Universal Robots PolyScope program: cobot_de_soudure_V2.2_GAPE.urp

Program cobot_de_soudure_V2.2_GAPE (installation=Cobot_de_soudure_V2.1_GAPE directory=/programs/Soudure 2023_03_27/V2.1 createdIn=5.9.4.1031232 lastSavedIn=5.11.9.1010452 robotSerialNumber=20225200921)
Calibrated DH parameters: a=[-0.00003, -0.368557, -0.560435, 0, -0.000026, 0]; d=[0.180818, -449.783649, 477.665205, -27.707784, 0.119652, 0.115612]; alpha=[1.571383, 0.001086, 0.003988, 1.568685, -1.571248, 0]; deltaTheta=[-0.000001, -0.924567, 7.403594, -0.195847, 0.000002, 0]
InitVariablesNode variables(variable(name=Test_Gaz, expression=False), variable(name=Test_Job, expression=False), variable(name=Test_Ordre_Mar, expression=False), variable(name=Valide_Gaz, expression=False), variable(name=fin_soud, expression=1), variable(name=secu_d, expression=0), variable(name=secu_g, expression=0), variable(name=timer_ret_gaz, expression=0))
BeforeStart
  Folder fonctions
    Folder Init [hidden by the author, left out]
    Folder Diverses
      Script file /programs/Soudure 2023_03_27/V2.1/scripts/Diverses/close_popup.script
        | #fermeture popup
        | 
        | def close_popup():
        | 	closepop = "close popup"
        |     	socket_send_string(closepop,"internal")
        |     	socket_send_byte(10,"internal")
        |     	socket_close()
        | 
        | 	closepop = "close popup"
        |     	socket_send_string(closepop,"internal")
        |     	socket_send_byte(10,"internal")
        |     	socket_close()
        | 	return(False)
        | end
      Script file /programs/Soudure 2023_03_27/V2.1/scripts/Diverses/debut_soud.script
        | def fun_debut_soudure():
        |     Valide_Gaz = False
        |     if  ((Test_Ordre_Mar == False) and (Test_Job == False)):
        |         Arc_On = True
        |         Test_Gaz = True
        |     end
        | end
      Script file /programs/Soudure 2023_03_27/V2.1/scripts/Diverses/fin_soudure.script
        | def fin_soudure():
        |         Arc_On = False
        |         Test_Gaz = False
        |         Test_Job = True
        |         Test_Ordre_Mar = True
        | end
      Script file /programs/Soudure 2023_03_27/V2.1/scripts/Diverses/fun_demande().script
        | #demande nombre soudures par type (compris entre 0 et 6)
        | 
        | def fun_demande(type):
        | 	if (1==type):
        | 		soudure = "point"					#si type = 1, la demande sera sur une soudure point
        | 	elif (2==type):
        | 		soudure = "lineaire"				#si type = 2, la demande sera sur une soudure linéaire
        | 	elif (3==type):
        | 		soudure = "arc de cercle"			#si type = 3, la demande sera sur une soudure arc de cercle
        | 	elif (4==type):
        | 		soudure = "cercle"					#si type = 4, la demande sera sur une soudure cercle
        | 	else :
        | 		return(False)
        | 	end
        | 
        | nb_soud = request_integer_from_primary_client("nombre de soudure(s) "+ soudure + " ?")			#la demande
        | 	if (nb_soud >6):																									#si la reponse est superieur a 6
        | 		popup1 = "popup le robot ne peut pas effectuer plus de 6 soudures "+ soudure + " sur la même pièce, réessayer."	#popup
        | 		socket_open("127.0.0.1",29999,"internal") # open internal socket
        | 
        | 		socket_send_line(popup1,"internal")         #Affichage Popup
        | 
        | 		socket_send_byte(10,"internal")
        | 		sleep(5.0)
        | 		closepop = "close popup"					#fermer popup
        | 		socket_send_string(closepop,"internal")
        | 		socket_send_byte(10,"internal")
        | 		socket_close()
        | 
        | 		while(nb_soud >6):
        | 			nb_soud = request_integer_from_primary_client("nombre de soudure(s) "+ soudure + " ? (compris entre 0 et 6 ;)")	#on redemande tant que le nombre est superieur a 6
        | 		end
        | end
        | return(nb_soud)        #on retourne le nombre de soudure à effectuer dans le type
        | end
      Script file /programs/Soudure 2023_03_27/V2.1/scripts/Diverses/fun_demande_job.script
        | #demande le job à utiliser (mode de soudure régler sur le poste à souder) (compris entre 0 et 3, pour 1 et 4 sur le poste a souder)
        | def fun_demande_job(type):
        | 	if (1==type):
        | 		soudure = "point"
        | 	elif (2==type):
        | 		soudure = "lineaire"
        | 	elif (3==type):
        | 		soudure = "arc de cercle"
        | 	elif (4==type):
        | 		soudure = "cercle"
        | 	else :
        | 		return(False)
        | 	end
        | 
        |   job = request_integer_from_primary_client("Mode du poste à souder pour soudure : "+ soudure + " ? [1-4]")
        |   job = job-1 #adapter la saisie aux besoins du code
        | 
        |   while ((job!=0) and (job!=1) and (job!=2) and (job!=3)): #reboucler si mauvaise saisie
        | 	  job = request_integer_from_primary_client("Mode du poste à souder pour soudure : "+ soudure + " ? [1-4]")
        |       job = job-1 #adapter la saisie aux besoins du code
        |   end
        | 
        | return(job)
        | end
      Script file /programs/Soudure 2023_03_27/V2.1/scripts/Diverses/fun_demande_type_soudure.script
        | #demande le type de soudure à enregistrer (entre 1 et 5)
        | def fun_demande_type_soudure():
        | 
        | 	reponse = request_integer_from_primary_client("1->POINT     2->LINEAIRE    3->ARC    4->CERCLE  5->FIN")
        | 
        |     if ((reponse == 0) or (reponse > 5)):
        |         reponse = 5
        |     end
        | 
        | return(reponse)
        | end
      Script file /programs/Soudure 2023_03_27/V2.1/scripts/Diverses/fun_demande_vit.script
        | #demande nombre soudures par type (compris entre 0 et 6)
        | def fun_demande_vit(type):
        | 	if (1==type):
        | 		soudure = "point"
        | 	elif (2==type):
        | 		soudure = "lineaire"
        | 	elif (3==type):
        | 		soudure = "arc de cercle"
        | 	elif (4==type):
        | 		soudure = "cercle"
        | 	else :
        | 		return(False)
        | 	end
        | 
        | vit_soud = request_float_from_primary_client("vitesse de la soudure "+ soudure + " ? (mm/s)")
        | 	#if (vit_soud >6):
        | 	#	popup1 = "popup le robot ne peut pas effectuer plus de 6 soudures "+ soudure + " sur la même pièce, réessayer."
        | 	#	socket_open("127.0.0.1",29999,"internal") # open internal socket
        | 
        | 	#	socket_send_line(popup1,"internal")         #Affichage Popup
        | 
        | 	#	socket_send_byte(10,"internal")
        | 	#	sleep(5.0)
        | 	#	closepop = "close popup"
        | 	#	socket_send_string(closepop,"internal")
        | 	#	socket_send_byte(10,"internal")
        | 	#	socket_close()
        | 
        | 	#	while(vit_soud >6):
        | 	#		vit_soud = request_integer_from_primary_client("nombre de soudure(s) "+ soudure + " ? (compris entre 0 et 6 ;)")
        | 	#	end
        | #end
        | return(vit_soud/1000)
        | end
      Script file /programs/Soudure 2023_03_27/V2.1/scripts/Diverses/fun_front_down.script
        | #attente front montant sur add_bp
        | 
        | def fun_front_do(add_bp):
        | bp = get_digital_in(add_bp)
        |     while not bp :
        |         bp = get_digital_in(add_bp)    #dans la boucle tant que l'entrée add_bp est a 1
        |         #attente relachement bouton
        |    end
        | 
        |     while bp :                              #dans la boucle tant que l'entrée add_bp est a 0
        |         bp = get_digital_in(add_bp)
        |         #attente
        |     end
        | 
        |     #while not bp :
        |            #bp = get_digital_in(add_bp)    #dans la boucle tant que l'entrée add_bp est a 1
        |      #end
        | 
        |     return(False)
        | end
      Script file /programs/Soudure 2023_03_27/V2.1/scripts/Diverses/fun_front_up.script
        | #attente front montant sur add_bp
        | 
        | def fun_front_up(add_bp):
        | bp = get_digital_in(add_bp)
        |     while bp :
        |         bp = get_digital_in(add_bp)    #dans la boucle tant que l'entrée add_bp est a 1
        |         #attente relachement bouton
        |     end
        | 
        |     while not bp :                              #dans la boucle tant que l'entrée add_bp est a 0
        |         bp = get_digital_in(add_bp)
        |         #attente
        |     end
        |     return(False)
        | end
      Script file /programs/Soudure 2023_03_27/V2.1/scripts/Diverses/fun_popup_soud().script
        | #ouvre un pop-up "configuration soudure (type_soud) n°(num_soud): placer le robot (etape_soud) et valider la position. (bp_cobot)". fermeture popup a l'aide de close_popup()
        | #pour la definition de la fonction :
        |     #etape :
        |     #   1 : approche
        |     #   2 : depart
        |     #   3 : premier quart
        |     #   4 : milieu
        |     #   5 : trois-quart
        |     #   6 : fin
        |     #   7 : retrait
        | 
        |     #type :
        |     #   1 : soudure point
        |     #   2 : soudure lineaire
        |     #   3 : soudure arc de cercle
        |     #   4 : soudure cercle
        |     #   5 : plus de soudure
        |     #num : i, j, k ou l correspondant au numero de la soudure ( i pour type = 1, j pour type = 2, k pour type = 3, l pour type = 4)
        | 
        | def fun_popup_soud(etape, type, num):
        | 
        |     switch_1 = etape
        |     switch_2 = type
        |         ##############################################################################
        | 
        |     ####################### POPUP-approche #######################################
        | 
        | ##############################################################################
        |     #switch etape
        |     if (1 == switch_1) : #point d'approche
        |         etape_soud = " en APPROCHE"
        |         #switch type
        |         if (1 == switch_2) : #soudure point
        |             type_soud = "point"
        | 
        |        elif (2 == switch_2) : #soudure lineaire
        |             type_soud = "lineaire"
        | 
        |         elif (3 == switch_2) : #soudure arc de cerlce
        |             type_soud = "arc de cercle"
        | 
        |         elif (4 == switch_2) : #soudure cercle
        |            type_soud = "cercle"
        | 
        |         else :
        |             return (False)
        |         end
        | 
        |         ##############################################################################
        | 
        |     ####################### POPUP-debut ##########################################
        | 
        | ##############################################################################
        | 
        |     elif (2 == switch_1): #point de soudure/debut
        |         #switch type
        |         if (1 == switch_2) : #soudure point
        |            etape_soud = "sur le POINT"
        |             type_soud = "point"
        | 
        |         elif (2 == switch_2): #soudure lineaire
        |             etape_soud = "sur le DEBUT"
        |             type_soud = "lineaire"
        | 
        |         elif (3 == switch_2) : #soudure arc de cerlce
        |             etape_soud = "sur le DEBUT"
        |             type_soud = "arc de cercle"
        | 
        |         elif (4 == switch_2) : #soudure cercle
        |             etape_soud = "sur le DEBUT"
        |            type_soud = "cercle"
        | 
        |         else :
        |             return (False)
        |         end
        | 
        |         ##############################################################################
        | 
        |     ####################### POPUP-quart ##########################################
        | 
        | ##############################################################################
        | 
        |     elif (3 == switch_1): #point de quart
        |         etape_soud = "sur 1er QUART"
        |         #switch type
        |         if (4 == switch_2) : #soudure cercle
        |             type_soud = "cercle"
        |         end
        | 
        |         ##############################################################################
        | 
        |     ####################### POPUP-milieu ########################################
        | 
        | #############################################################################
        | 
        |     elif (4 == switch_1): #point de milieu
        |         etape_soud = "à la MOITIE"
        |         #switch type
        |         if (3 == switch_2) : #soudure arc de cercle
        |             type_soud = "arc de cercle"
        |         elif (4 == switch_2): #soudure arc de cercle
        |             type_soud = "cercle"
        |         end
        | 
        |         ##############################################################################
        | 
        |     ####################### POPUP-trois_quart ####################################
        | 
        | ##############################################################################
        | 
        |     elif (5 == switch_1): #point trois_quart
        |         etape_soud = "sur le 3e QUART"
        |         #switch type
        |         if (4 == switch_2) : #soudure cercle
        |             type_soud = "cercle"
        |         end
        | 
        |         ##############################################################################
        | 
        |     ####################### POPUP-fin ############################################
        | 
        | ##############################################################################
        | 
        |     elif (6 == switch_1): #point de fin
        |         etape_soud = "sur la FIN"
        |         #switch type
        |         if (2 == switch_2) : #soudure lineaire
        |             type_soud = "lineaire"
        | 
        |         elif (3 == switch_2) : #soudure arc de cerlce
        |             type_soud = "arc de cercle"
        | 
        |         elif (4 == switch_2) : #soudure cercle
        |             type_soud = "cercle"
        | 
        |         else :
        |             return (False)
        |         end
        | 
        |         ##############################################################################
        | 
        |     ####################### POPUP-retrait ########################################
        | 
        | ##############################################################################
        | 
        |     elif (7 == switch_1): #point de retrait
        |         etape_soud = "en RETRAIT"
        |         #switch type
        |         if (2 == switch_2) : #soudure lineaire
        |             type_soud = "lineaire"
        | 
        |         elif (3 == switch_2) : #soudure arc de cerlce
        |            type_soud = "arc de cercle"
        | 
        |         elif (4 == switch_2) : #soudure cercle
        |            type_soud = "cercle"
        | 
        |         else :
        |            return (False)
        |         end
        | 
        |     else :
        |         return(False)
        |     end
        | 
        |         ##############################################################################
        | 
        |     ######################## affichage_POPUP #####################################
        | 
        | ##############################################################################
        |     sync()
        |     num_soud = to_str(num)
        |     popup1 = "popup Config. : " + type_soud + " n°" + num_soud + " : placer " + etape_soud + " & Valider"             #on ouvre un popup
        |     socket_open("127.0.0.1",29999,"internal") # open internal socket
        |     socket_send_line(popup1,"internal")     #Affichage message
        |     socket_send_byte(10,"internal")
        |     sync()
        | end
      Script file /programs/Soudure 2023_03_27/V2.1/scripts/Diverses/fun_raz_d.script
        | def fun_raz_d():
        |     #taille des tableaux de positions = nombre de soudures maximum par type + 1 (car commence à enregistrer à l'index 1)
        |     global tab_point_app_d =    [p[0,0,0,0,0,0], p[0,0,0,0,0,0], p[0,0,0,0,0,0], p[0,0,0,0,0,0], p[0,0,0,0,0,0], p[0,0,0,0,0,0], p[0,0,0,0,0,0], p[0,0,0,0,0,0], p[0,0,0,0,0,0], p[0,0,0,0,0,0], p[0,0,0,0,0,0]]
        |     global tab_point_deb_d =    [p[0,0,0,0,0,0], p[0,0,0,0,0,0], p[0,0,0,0,0,0], p[0,0,0,0,0,0], p[0,0,0,0,0,0], p[0,0,0,0,0,0], p[0,0,0,0,0,0], p[0,0,0,0,0,0], p[0,0,0,0,0,0], p[0,0,0,0,0,0], p[0,0,0,0,0,0]]
        |     global tab_point_ret_d =    [p[0,0,0,0,0,0], p[0,0,0,0,0,0], p[0,0,0,0,0,0], p[0,0,0,0,0,0], p[0,0,0,0,0,0], p[0,0,0,0,0,0], p[0,0,0,0,0,0], p[0,0,0,0,0,0], p[0,0,0,0,0,0], p[0,0,0,0,0,0], p[0,0,0,0,0,0]]
        | 
        |     global tab_lin_app_d =      [p[0,0,0,0,0,0], p[0,0,0,0,0,0], p[0,0,0,0,0,0], p[0,0,0,0,0,0], p[0,0,0,0,0,0], p[0,0,0,0,0,0], p[0,0,0,0,0,0], p[0,0,0,0,0,0], p[0,0,0,0,0,0], p[0,0,0,0,0,0], p[0,0,0,0,0,0]]
        |     global tab_lin_deb_d =      [p[0,0,0,0,0,0], p[0,0,0,0,0,0], p[0,0,0,0,0,0], p[0,0,0,0,0,0], p[0,0,0,0,0,0], p[0,0,0,0,0,0], p[0,0,0,0,0,0], p[0,0,0,0,0,0], p[0,0,0,0,0,0], p[0,0,0,0,0,0], p[0,0,0,0,0,0]]
        |     global tab_lin_fin_d =      [p[0,0,0,0,0,0], p[0,0,0,0,0,0], p[0,0,0,0,0,0], p[0,0,0,0,0,0], p[0,0,0,0,0,0], p[0,0,0,0,0,0], p[0,0,0,0,0,0], p[0,0,0,0,0,0], p[0,0,0,0,0,0], p[0,0,0,0,0,0], p[0,0,0,0,0,0]]
        |     global tab_lin_ret_d =      [p[0,0,0,0,0,0], p[0,0,0,0,0,0], p[0,0,0,0,0,0], p[0,0,0,0,0,0], p[0,0,0,0,0,0], p[0,0,0,0,0,0], p[0,0,0,0,0,0], p[0,0,0,0,0,0], p[0,0,0,0,0,0], p[0,0,0,0,0,0], p[0,0,0,0,0,0]]
        | 
        |     global tab_arc_app_d =      [p[0,0,0,0,0,0], p[0,0,0,0,0,0], p[0,0,0,0,0,0], p[0,0,0,0,0,0], p[0,0,0,0,0,0], p[0,0,0,0,0,0], p[0,0,0,0,0,0], p[0,0,0,0,0,0], p[0,0,0,0,0,0], p[0,0,0,0,0,0], p[0,0,0,0,0,0]]
        |     global tab_arc_deb_d =      [p[0,0,0,0,0,0], p[0,0,0,0,0,0], p[0,0,0,0,0,0], p[0,0,0,0,0,0], p[0,0,0,0,0,0], p[0,0,0,0,0,0], p[0,0,0,0,0,0], p[0,0,0,0,0,0], p[0,0,0,0,0,0], p[0,0,0,0,0,0], p[0,0,0,0,0,0]]
        |     global tab_arc_mil_d =      [p[0,0,0,0,0,0], p[0,0,0,0,0,0], p[0,0,0,0,0,0], p[0,0,0,0,0,0], p[0,0,0,0,0,0], p[0,0,0,0,0,0], p[0,0,0,0,0,0], p[0,0,0,0,0,0], p[0,0,0,0,0,0], p[0,0,0,0,0,0], p[0,0,0,0,0,0]]
        |     global tab_arc_fin_d =      [p[0,0,0,0,0,0], p[0,0,0,0,0,0], p[0,0,0,0,0,0], p[0,0,0,0,0,0], p[0,0,0,0,0,0], p[0,0,0,0,0,0], p[0,0,0,0,0,0], p[0,0,0,0,0,0], p[0,0,0,0,0,0], p[0,0,0,0,0,0], p[0,0,0,0,0,0]]
        |     global tab_arc_ret_d =      [p[0,0,0,0,0,0], p[0,0,0,0,0,0], p[0,0,0,0,0,0], p[0,0,0,0,0,0], p[0,0,0,0,0,0], p[0,0,0,0,0,0], p[0,0,0,0,0,0], p[0,0,0,0,0,0], p[0,0,0,0,0,0], p[0,0,0,0,0,0], p[0,0,0,0,0,0]]
        | 
        |     global tab_cer_app_d =      [p[0,0,0,0,0,0], p[0,0,0,0,0,0], p[0,0,0,0,0,0], p[0,0,0,0,0,0], p[0,0,0,0,0,0], p[0,0,0,0,0,0], p[0,0,0,0,0,0], p[0,0,0,0,0,0], p[0,0,0,0,0,0], p[0,0,0,0,0,0], p[0,0,0,0,0,0]]
        |     global tab_cer_deb_d =      [p[0,0,0,0,0,0], p[0,0,0,0,0,0], p[0,0,0,0,0,0], p[0,0,0,0,0,0], p[0,0,0,0,0,0], p[0,0,0,0,0,0], p[0,0,0,0,0,0], p[0,0,0,0,0,0], p[0,0,0,0,0,0], p[0,0,0,0,0,0], p[0,0,0,0,0,0]]
        |     global tab_cer_quart_d =    [p[0,0,0,0,0,0], p[0,0,0,0,0,0], p[0,0,0,0,0,0], p[0,0,0,0,0,0], p[0,0,0,0,0,0], p[0,0,0,0,0,0], p[0,0,0,0,0,0], p[0,0,0,0,0,0], p[0,0,0,0,0,0], p[0,0,0,0,0,0], p[0,0,0,0,0,0]]
        |     global tab_cer_mil_d =      [p[0,0,0,0,0,0], p[0,0,0,0,0,0], p[0,0,0,0,0,0], p[0,0,0,0,0,0], p[0,0,0,0,0,0], p[0,0,0,0,0,0], p[0,0,0,0,0,0], p[0,0,0,0,0,0], p[0,0,0,0,0,0], p[0,0,0,0,0,0], p[0,0,0,0,0,0]]
        |     global tab_cer_tro_d =      [p[0,0,0,0,0,0], p[0,0,0,0,0,0], p[0,0,0,0,0,0], p[0,0,0,0,0,0], p[0,0,0,0,0,0], p[0,0,0,0,0,0], p[0,0,0,0,0,0], p[0,0,0,0,0,0], p[0,0,0,0,0,0], p[0,0,0,0,0,0], p[0,0,0,0,0,0]]
        |     global tab_cer_fin_d =      [p[0,0,0,0,0,0], p[0,0,0,0,0,0], p[0,0,0,0,0,0], p[0,0,0,0,0,0], p[0,0,0,0,0,0], p[0,0,0,0,0,0], p[0,0,0,0,0,0], p[0,0,0,0,0,0], p[0,0,0,0,0,0], p[0,0,0,0,0,0], p[0,0,0,0,0,0]]
        |     global tab_cer_ret_d =      [p[0,0,0,0,0,0], p[0,0,0,0,0,0], p[0,0,0,0,0,0], p[0,0,0,0,0,0], p[0,0,0,0,0,0], p[0,0,0,0,0,0], p[0,0,0,0,0,0], p[0,0,0,0,0,0], p[0,0,0,0,0,0], p[0,0,0,0,0,0], p[0,0,0,0,0,0]]
        | 
        |      #2 nouveaux tableaux modif V2.1 (longueur 40 si 4(type)*10(nb soudures max par type) ) -> mis 45 (permettre décalage + marge)
        |     global tab_type_d = [0,0,0,0,0,0,0,0,0,0,0,0,0,0,0,0,0,0,0,0,0,0,0,0,0,0,0,0,0,0,0,0,0,0,0,0,0,0,0,0,0,0,0,0,0]
        |     global tab_job_d  = [0,0,0,0,0,0,0,0,0,0,0,0,0,0,0,0,0,0,0,0,0,0,0,0,0,0,0,0,0,0,0,0,0,0,0,0,0,0,0,0,0,0,0,0,0]
        | 
        |     #vitesses de soudure
        |     global tps_point_d = 0
        |     global vit_arc_d = [0,0,0,0,0,0,0,0,0,0,0]
        |     global vit_cer_d = [0,0,0,0,0,0,0,0,0,0,0]
        |     global vit_lin_d = [0,0,0,0,0,0,0,0,0,0,0]
        | 
        |     global nb_soud_point_d  = 0
        |     global nb_soud_lin_d    = 0
        |     global nb_soud_arc_d    = 0
        |     global nb_soud_cer_d    = 0
        | 
        |     global nbSoudure_glo_d  = 0
        | 
        | end
      Script file /programs/Soudure 2023_03_27/V2.1/scripts/Diverses/fun_raz_g.script
        | def fun_raz_g():
        |     #taille des tableaux de positions = nombre de soudures maximum par type + 1 (car commence à enregistrer à l'index 1)
        |     global tab_point_app_g =    [p[0,0,0,0,0,0], p[0,0,0,0,0,0], p[0,0,0,0,0,0], p[0,0,0,0,0,0], p[0,0,0,0,0,0], p[0,0,0,0,0,0], p[0,0,0,0,0,0], p[0,0,0,0,0,0], p[0,0,0,0,0,0], p[0,0,0,0,0,0], p[0,0,0,0,0,0]]
        |     global tab_point_deb_g =    [p[0,0,0,0,0,0], p[0,0,0,0,0,0], p[0,0,0,0,0,0], p[0,0,0,0,0,0], p[0,0,0,0,0,0], p[0,0,0,0,0,0], p[0,0,0,0,0,0], p[0,0,0,0,0,0], p[0,0,0,0,0,0], p[0,0,0,0,0,0], p[0,0,0,0,0,0]]
        |     global tab_point_ret_g =    [p[0,0,0,0,0,0], p[0,0,0,0,0,0], p[0,0,0,0,0,0], p[0,0,0,0,0,0], p[0,0,0,0,0,0], p[0,0,0,0,0,0], p[0,0,0,0,0,0], p[0,0,0,0,0,0], p[0,0,0,0,0,0], p[0,0,0,0,0,0], p[0,0,0,0,0,0]]
        | 
        |     global tab_lin_app_g =      [p[0,0,0,0,0,0], p[0,0,0,0,0,0], p[0,0,0,0,0,0], p[0,0,0,0,0,0], p[0,0,0,0,0,0], p[0,0,0,0,0,0], p[0,0,0,0,0,0], p[0,0,0,0,0,0], p[0,0,0,0,0,0], p[0,0,0,0,0,0], p[0,0,0,0,0,0]]
        |     global tab_lin_deb_g =      [p[0,0,0,0,0,0], p[0,0,0,0,0,0], p[0,0,0,0,0,0], p[0,0,0,0,0,0], p[0,0,0,0,0,0], p[0,0,0,0,0,0], p[0,0,0,0,0,0], p[0,0,0,0,0,0], p[0,0,0,0,0,0], p[0,0,0,0,0,0], p[0,0,0,0,0,0]]
        |     global tab_lin_fin_g =      [p[0,0,0,0,0,0], p[0,0,0,0,0,0], p[0,0,0,0,0,0], p[0,0,0,0,0,0], p[0,0,0,0,0,0], p[0,0,0,0,0,0], p[0,0,0,0,0,0], p[0,0,0,0,0,0], p[0,0,0,0,0,0], p[0,0,0,0,0,0], p[0,0,0,0,0,0]]
        |     global tab_lin_ret_g =      [p[0,0,0,0,0,0], p[0,0,0,0,0,0], p[0,0,0,0,0,0], p[0,0,0,0,0,0], p[0,0,0,0,0,0], p[0,0,0,0,0,0], p[0,0,0,0,0,0], p[0,0,0,0,0,0], p[0,0,0,0,0,0], p[0,0,0,0,0,0], p[0,0,0,0,0,0]]
        | 
        |     global tab_arc_app_g =      [p[0,0,0,0,0,0], p[0,0,0,0,0,0], p[0,0,0,0,0,0], p[0,0,0,0,0,0], p[0,0,0,0,0,0], p[0,0,0,0,0,0], p[0,0,0,0,0,0], p[0,0,0,0,0,0], p[0,0,0,0,0,0], p[0,0,0,0,0,0], p[0,0,0,0,0,0]]
        |     global tab_arc_deb_g =      [p[0,0,0,0,0,0], p[0,0,0,0,0,0], p[0,0,0,0,0,0], p[0,0,0,0,0,0], p[0,0,0,0,0,0], p[0,0,0,0,0,0], p[0,0,0,0,0,0], p[0,0,0,0,0,0], p[0,0,0,0,0,0], p[0,0,0,0,0,0], p[0,0,0,0,0,0]]
        |     global tab_arc_mil_g =      [p[0,0,0,0,0,0], p[0,0,0,0,0,0], p[0,0,0,0,0,0], p[0,0,0,0,0,0], p[0,0,0,0,0,0], p[0,0,0,0,0,0], p[0,0,0,0,0,0], p[0,0,0,0,0,0], p[0,0,0,0,0,0], p[0,0,0,0,0,0], p[0,0,0,0,0,0]]
        |     global tab_arc_fin_g =      [p[0,0,0,0,0,0], p[0,0,0,0,0,0], p[0,0,0,0,0,0], p[0,0,0,0,0,0], p[0,0,0,0,0,0], p[0,0,0,0,0,0], p[0,0,0,0,0,0], p[0,0,0,0,0,0], p[0,0,0,0,0,0], p[0,0,0,0,0,0], p[0,0,0,0,0,0]]
        |     global tab_arc_ret_g =      [p[0,0,0,0,0,0], p[0,0,0,0,0,0], p[0,0,0,0,0,0], p[0,0,0,0,0,0], p[0,0,0,0,0,0], p[0,0,0,0,0,0], p[0,0,0,0,0,0], p[0,0,0,0,0,0], p[0,0,0,0,0,0], p[0,0,0,0,0,0], p[0,0,0,0,0,0]]
        | 
        |     global tab_cer_app_g =      [p[0,0,0,0,0,0], p[0,0,0,0,0,0], p[0,0,0,0,0,0], p[0,0,0,0,0,0], p[0,0,0,0,0,0], p[0,0,0,0,0,0], p[0,0,0,0,0,0], p[0,0,0,0,0,0], p[0,0,0,0,0,0], p[0,0,0,0,0,0], p[0,0,0,0,0,0]]
        |     global tab_cer_deb_g =      [p[0,0,0,0,0,0], p[0,0,0,0,0,0], p[0,0,0,0,0,0], p[0,0,0,0,0,0], p[0,0,0,0,0,0], p[0,0,0,0,0,0], p[0,0,0,0,0,0], p[0,0,0,0,0,0], p[0,0,0,0,0,0], p[0,0,0,0,0,0], p[0,0,0,0,0,0]]
        |     global tab_cer_quart_g =    [p[0,0,0,0,0,0], p[0,0,0,0,0,0], p[0,0,0,0,0,0], p[0,0,0,0,0,0], p[0,0,0,0,0,0], p[0,0,0,0,0,0], p[0,0,0,0,0,0], p[0,0,0,0,0,0], p[0,0,0,0,0,0], p[0,0,0,0,0,0], p[0,0,0,0,0,0]]
        |     global tab_cer_mil_g =      [p[0,0,0,0,0,0], p[0,0,0,0,0,0], p[0,0,0,0,0,0], p[0,0,0,0,0,0], p[0,0,0,0,0,0], p[0,0,0,0,0,0], p[0,0,0,0,0,0], p[0,0,0,0,0,0], p[0,0,0,0,0,0], p[0,0,0,0,0,0], p[0,0,0,0,0,0]]
        |     global tab_cer_tro_g =      [p[0,0,0,0,0,0], p[0,0,0,0,0,0], p[0,0,0,0,0,0], p[0,0,0,0,0,0], p[0,0,0,0,0,0], p[0,0,0,0,0,0], p[0,0,0,0,0,0], p[0,0,0,0,0,0], p[0,0,0,0,0,0], p[0,0,0,0,0,0], p[0,0,0,0,0,0]]
        |     global tab_cer_fin_g =      [p[0,0,0,0,0,0], p[0,0,0,0,0,0], p[0,0,0,0,0,0], p[0,0,0,0,0,0], p[0,0,0,0,0,0], p[0,0,0,0,0,0], p[0,0,0,0,0,0], p[0,0,0,0,0,0], p[0,0,0,0,0,0], p[0,0,0,0,0,0], p[0,0,0,0,0,0]]
        |     global tab_cer_ret_g =      [p[0,0,0,0,0,0], p[0,0,0,0,0,0], p[0,0,0,0,0,0], p[0,0,0,0,0,0], p[0,0,0,0,0,0], p[0,0,0,0,0,0], p[0,0,0,0,0,0], p[0,0,0,0,0,0], p[0,0,0,0,0,0], p[0,0,0,0,0,0], p[0,0,0,0,0,0]]
        | 
        |      #2 nouveaux tableaux modif V2.1 (longueur 40 si 4(type)*10(nb soudures max par type) ) -> mis 45 (permettre décalage + marge)
        |     global tab_type_g = [0,0,0,0,0,0,0,0,0,0,0,0,0,0,0,0,0,0,0,0,0,0,0,0,0,0,0,0,0,0,0,0,0,0,0,0,0,0,0,0,0,0,0,0,0]
        |     global tab_job_g  = [0,0,0,0,0,0,0,0,0,0,0,0,0,0,0,0,0,0,0,0,0,0,0,0,0,0,0,0,0,0,0,0,0,0,0,0,0,0,0,0,0,0,0,0,0]
        | 
        |     #vitesses de soudure
        |     global tps_point_g = 0
        |     global vit_arc_g = [0,0,0,0,0,0,0,0,0,0,0]
        |     global vit_cer_g = [0,0,0,0,0,0,0,0,0,0,0]
        |     global vit_lin_g = [0,0,0,0,0,0,0,0,0,0,0]
        | 
        |     global nb_soud_point_g  = 0
        |     global nb_soud_lin_g    = 0
        |     global nb_soud_arc_g    = 0
        |     global nb_soud_cer_g    = 0
        | 
        |     global nbSoudure_glo_g  = 0
        | end
    Folder Demande
      Script file /programs/Soudure 2023_03_27/V2.1/scripts/Demande/demande_d.script
        | def fun_demande_d():
        | 
        |     close_popup()
        |     nb_soud_point_d = fun_demande(1)
        |     if (nb_soud_point_d > 0):
        |             tps_point_d = request_float_from_primary_client("temps des soudures points ? (s)")
        |     end
        |     nb_soud_lin_d = fun_demande(2)
        |     nb_soud_arc_d = fun_demande(3)
        |     nb_soud_cer_d = fun_demande(4)
        | 
        | end
      Script file /programs/Soudure 2023_03_27/V2.1/scripts/Demande/demande_g.script
        | def fun_demande_g():
        |      close_popup()
        |      nb_soud_point_g = fun_demande(1)
        |      nb_soud_lin_g = fun_demande(2)
        |      if nb_soud_lin_g > 0:
        |           vit_lin_g = fun_demande_vit(2)
        |      end
        |      nb_soud_arc_g = fun_demande(3)
        |      if nb_soud_arc_g > 0:
        |           vit_arc_g = fun_demande_vit(3)
        |      end
        |      nb_soud_cer_g = fun_demande(4)
        |      if nb_soud_arc_g > 0:
        |           vit_cer_g = fun_demande_vit(4)
        |      end
        | end
    Folder Configuration [hidden by the author, left out]
    Folder Execution
      Script file /programs/Soudure 2023_03_27/V2.1/scripts/Execution/execution_d.script
        | def fun_execution_d():
        |     ######################## INITIALISATION #########################################
        |     #adressage
        |     adresse_bp_cobot = 2                                    #adresse cobot bp_cobot
        |     adresse_bp_d = 3                                        #adresse cobot bp_g
        | #VARIABLES CI DESSUS UTILES ?????
        | 
        | 
        |     local index_soudure_point = 1
        |     local index_soudure_lin = 1
        |     local index_soudure_arc = 1
        |     local index_soudure_cer = 1
        | 
        |     close_popup()
        |     #config popup
        |     popup1 = "popup Table droite, éxécution..."
        |     socket_open("127.0.0.1",29999,"internal")
        |     socket_send_line(popup1,"internal")
        |     socket_send_byte(10,"internal")
        | 
        |     fun_deplacement_pose_inter(2)    #deplacement dans la position intermédiaire enregistrée
        | 
        |     local nbSoudures = nbSoudure_glo_d
        |     local soudureEnCours = 0 #soudure en cours
        |     local job = 0
        |     local typeSoudure = 0
        | 
        |     while (soudureEnCours<nbSoudures): #pour le moment début a 0 donc < (a voir si changement necessaire)
        |         job = tab_job_d[soudureEnCours]
        |         fun_commande_job(job)
        |         typeSoudure = tab_type_d[soudureEnCours]
        | 
        |         #switch de tous les types avec appel aux fonctions correspondantes
        |         if (typeSoudure == 1 ):
        |             fun_soudure_point(index_soudure_point,2) # ( , 2 pour signifier table de droite )
        |             #fun_soudure_point(index_soudure_point)
        |             index_soudure_point = index_soudure_point + 1
        |         elif (typeSoudure == 2 ):
        |             fun_soudure_lineaire(index_soudure_lin,2)
        |             index_soudure_lin = index_soudure_lin + 1
        |         elif (typeSoudure == 3 ):
        |             fun_soudure_arc(index_soudure_arc,2)
        |             index_soudure_arc = index_soudure_arc +1
        |         elif (typeSoudure == 4 ):
        |             fun_soudure_cercle(index_soudure_cercle,2)
        |             index_soudure_cercle = index_soudure_cercle +1
        |         else:
        |         end
        |         soudureEnCours = soudureEnCours +1
        |         sync()
        |     end
        |         #movej(anti_poq_d_1, a=1.4,v=1.1,t=0,r=0.005)
        |         #movej(anti_poq_d_2, a=1.4,v=1.1,t=0,r=0.005)
        |         movej(Point_Attente_D, a=0.8,v=1.05,t=0,r=0.005)
        |         movej(Point_init_D, a=0.8,v=1.05,t=0,r=0.005)
        |         movej(Point_avt_initD, a=0.8,v=1.05,t=0,r=0.005)
        |         movej(Point_init, a=0.8,v=1.05,t=0,r=0)
        | end
      Script file /programs/Soudure 2023_03_27/V2.1/scripts/Execution/execution_g.script
        | def fun_execution_g():
        | ######################## INITIALISATION #######################################
        | 
        | #adressage
        | adresse_bp_cobot = 2                                    #adresse cobot bp_cobot
        | adresse_bp_g = 2                                        #adresse cobot bp_g
        | #VARIABLES CI DESSUS UTILES ?????
        | 
        | 
        | local index_soudure_point = 1
        | local index_soudure_lin = 1
        | local index_soudure_arc = 1
        | local index_soudure_cer = 1
        | 
        | close_popup()
        | #config popup
        | #popup1 = "popup Table gauche, éxécution..."
        | #socket_open("127.0.0.1",29999,"internal")
        | #socket_send_line(popup1,"internal")
        | #socket_send_byte(10,"internal")
        | 
        | #fun_deplacement_pose_inter(1)
        | 
        | local nbSoudures = nbSoudure_glo_g
        | local soudureEnCours = 0 #soudure en cours
        | local job = 0
        | local typeSoudure = 0
        | 
        | while (soudureEnCours<nbSoudures): #pour le moment début a 0 donc < (a voir si changement necessaire)
        |     job = tab_job_g[soudureEnCours]
        |     fun_commande_job(job)
        |     typeSoudure = tab_type_g[soudureEnCours]
        | 
        |     #switch de tous les types avec appel aux fonctions correspondantes
        |     if (typeSoudure == 1 ):
        |         #fun_soudure_point(index_soudure_point)
        |         fun_soudure_point(index_soudure_point,1) # ( , 1 pour signifier table de gauche )
        |         index_soudure_point = index_soudure_point + 1
        |     elif (typeSoudure == 2 ):
        |         fun_soudure_lineaire(index_soudure_lin,1)
        |         index_soudure_lin = index_soudure_lin + 1
        |     elif (typeSoudure == 3 ):
        |         fun_soudure_arc(index_soudure_arc,1)
        |         index_soudure_arc = index_soudure_arc +1
        |     elif (typeSoudure == 4 ):
        |         fun_soudure_cercle(index_soudure_cercle,1)
        |         index_soudure_cercle = index_soudure_cercle +1
        |     else:
        |     end
        |     soudureEnCours = soudureEnCours +1
        |     sync()
        | end
        |     #movej(anti_Poq_g, a=1.4,v=1.1,t=0,r=0.005)
        |     #movej(Point_init, a=1.4,v=1.1,t=0,r=0.005)
        | 
        |    # movej(Point_Attente_G, a=0.8,v=1.05,t=0,r=0.005)
        |     #movej(Point_init_G, a=0.8,v=1.05,t=0,r=0.005)
        |    # movej(Point_init, a=0.8,v=1.05,t=0,r=0)
        | 
        | end
      Script file /programs/Soudure 2023_03_27/V2.1/scripts/Execution/fun_activer_soudure.script
        | def fun_activer_soudure():
        |     soudure_on = 1
        |     sleep(tps_init_soud)
        |     sync()
        | end
      Script file /programs/Soudure 2023_03_27/V2.1/scripts/Execution/fun_fin_soudure.script
        | def fun_fin_soudure(table):
        | 
        |     soudure_on = 0
        |     while(fin_soud == 0):
        |     end
        |     set_digital_out(table+4,False)                 #eteindre la lumiere pour dire que l'on soude plus
        | 
        |     #table +4 : les sorties numériques sont respectivements 5 table gauche & 6 table droite
        |     #le décalage permet d'écrire directement au bon endroit
        |     sync()
        | 
        | end
      Script file /programs/Soudure 2023_03_27/V2.1/scripts/Execution/fun_commande_job.script
        | #fonction ecriture des jobs vers rob3000
        | def fun_commande_job(int):
        | 
        |     if (int == 0):
        |         set_digital_out(2,False)
        |         set_digital_out(3,False)
        | 
        | 
        |     elif(int == 1):
        |         set_digital_out(2,True)
        |         set_digital_out(3,False)
        | 
        |     elif(int == 2):
        |         set_digital_out(2,False)
        |         set_digital_out(3,True)
        | 
        |     elif(int == 3):
        |         set_digital_out(2,True)
        |         set_digital_out(3,True)
        | 
        |    # else:
        |    #     set_digital_out(2,False)
        |      #   set_digital_out(3,False)
        |     end
        | end
      Script file /programs/Soudure 2023_03_27/V2.1/scripts/Execution/fun_deplacement_pose_inter.script
        | def fun_deplacement_pose_inter(table):
        |     a_fun = 0.2
        |     v_fun = 1.1
        |     r_fun= 0
        |     t_fun = 0
        |     if (table == 1): #si 1 -> Table de gauche
        |       #  movej(pose_inter_g,a=a_fun,v=v_fun,t=t_fun,r=r_fun)
        |     else: #sinon table de droite
        |      #   movej(pose_inter_d,a=a_fun,v=v_fun,t=t_fun,r=r_fun)
        |     end
        |     sync()
        | end
      Script file /programs/Soudure 2023_03_27/V2.1/scripts/Execution/fun_soudure_arc.script
        | def fun_soudure_arc(Index,table):
        |     a_fun = 0.5
        |     v_fun = 1.1
        |     r_fun= 0.00
        |     t_fun = 0
        |     if (table == 1): #si 1 -> Table de gauche
        | 
        |         movej(tab_arc_app_g[Index],a_fun,v=v_fun,t=t_fun,r=r_fun)
        |         set_digital_out(5,True)                     #Allumer la lumiere pour dire que l'on soude
        |         movej(tab_arc_deb_g[Index],a_fun,v=v_fun,t=t_fun,r=r_fun)
        | 
        |         fun_activer_soudure()                        #appel de la fonction activer la soudure
        | 
        |         movec(tab_arc_mil_g[Index], tab_arc_fin_g[Index], a_fun,v=vit_arc_g[Index], r=0.002)
        | 
        |         fun_fin_soudure(1)                           #appel de la fonction désactiver la soudure
        | 
        |         movej(tab_arc_ret_g[Index],a=a_fun,v=v_fun,t=t_fun,r=r_fun)
        | 
        |         fun_deplacement_pose_inter(1)                     #appel de la fonction de déplacement en pose intermédiaire
        | 
        |     else: #sinon table de droite
        | 
        |         movej(tab_arc_app_d[Index],a_fun,v=v_fun,t=t_fun,r=r_fun)
        |         set_digital_out(6,True)                     #Allumer la lumiere pour dire que l'on soude
        |         movej(tab_arc_deb_d[Index],a_fun,v=v_fun,t=t_fun,r =r_fun)
        | 
        |         fun_activer_soudure()                        #appel de la fonction activer la soudure
        | 
        |         movec(tab_arc_mil_d[Index], tab_arc_fin_d[Index], a_fun,v=vit_arc_d[Index], r=0.002)
        | 
        |         fun_fin_soudure(2)                           #appel de la fonction désactiver la soudure
        | 
        |         movej(tab_arc_ret_d[Index],a_fun,v=v_fun,t=t_fun,r=r_fun)
        | 
        |         fun_deplacement_pose_inter(2)                     #appel de la fonction de déplacement en pose intermédiaire
        |     end
        |     sync()
        | end
      Script file /programs/Soudure 2023_03_27/V2.1/scripts/Execution/fun_soudure_cercle.script
        | def fun_soudure_cercle(Index,table):
        |     a_fun = 0.5
        |     v_fun = 1.1
        |     r_fun= 0.0
        |     t_fun = 0
        |     if (table == 1): #si 1 -> Table de gauche
        |         movej(tab_cer_app_g[Index],a=a_fun,v=v_fun,t=t_fun,r=r_fun)
        |         set_digital_out(5,True)                     #Allumer la lumiere pour dire que l'on soude
        |         movej(tab_cer_deb_g[Index],a=a_fun,v=v_fun,t=t_fun,r=r_fun)
        | 
        |         fun_activer_soudure()                        #appel de la fonction activer la soudure
        | 
        |         movec(tab_cer_quart_g[Index], tab_cer_mil_g[Index], a=a_fun,v=vit_cer_g[Index], r=0.002)
        |         movec(tab_cer_tro_g[Index], tab_cer_fin_g[Index], a=a_fun,v=vit_cer_g[Index], r=0.002)
        | 
        |         fun_fin_soudure(1)                           #appel de la fonction désactiver la soudure
        | 
        |         movej(tab_cer_ret_g[Index],a=a_fun, v=v_fun, t=t_fun, r=r_fun)
        | 
        |         fun_deplacement_pose_inter(1)                     #appel de la fonction de déplacement en pose intermédiaire
        | 
        |     else: #sinon table de droite
        |         movej(tab_cer_app_d[Index],a=a_fun,v=v_fun,t=t_fun,r=r_fun)
        |         set_digital_out(6,True)                     #Allumer la lumiere pour dire que l'on soude
        |         movej(tab_cer_deb_d[Index],a=a_fun,v=v_fun,t=t_fun,r=r_fun)
        | 
        |         fun_activer_soudure()                       #appel de la fonction activer la soudure
        | 
        |         movec(tab_cer_quart_d[Index], tab_cer_mil_d[Index], a=a_fun,v=vit_cer_d[Index], r=0.002)
        |         movec(tab_cer_tro_d[Index], tab_cer_fin_d[Index], a=a_fun, v=vit_cer_d[Index], r=0.002)
        | 
        |         fun_fin_soudure(2)                           #appel de la fonction désactiver la soudure
        | 
        |         movej(tab_cer_ret_d[Index],a=a_fun, v=v_fun, t=t_fun, r=r_fun)
        | 
        |         fun_deplacement_pose_inter(2)                     #appel de la fonction de déplacement en pose intermédiaire
        | 
        |     end
        |     sync()
        | end
      Script file /programs/Soudure 2023_03_27/V2.1/scripts/Execution/fun_soudure_lineaire.script
        | def fun_soudure_lineaire(Index,table):
        |     a_fun = 2
        |     v_fun = 4
        |     r_fun= 0.00
        |     t_fun = 0
        |     if (table == 1): #si 1 -> Table de gauche
        |         movej(tab_lin_app_g[Index],a=a_fun,v=v_fun,t=t_fun,r=r_fun)
        |         set_digital_out(5,True)                     #Allumer la lumiere pour dire que l'on soude
        |         movej(tab_lin_deb_g[Index],a=a_fun,v=v_fun,t=t_fun,r=r_fun)
        | 
        |         fun_activer_soudure()                         #appel de la fonction activer la soudure
        | 
        |         movel(tab_lin_fin_g[Index],a=a_fun,v=vit_lin_g[Index],t=t_fun)
        | 
        |         fun_fin_soudure(1)                           #appel de la fonction désactiver la soudure
        | 
        |         movej(tab_lin_ret_g[Index],a=a_fun,v=v_fun,t=t_fun,r=r_fun)
        | 
        |         fun_deplacement_pose_inter(1)                     #appel de la fonction de déplacement en pose intermédiaire
        | 
        | 
        |     else: #sinon table de droite
        | 
        |         movej(tab_lin_app_d[Index],a=a_fun,v=v_fun,t=t_fun,r=r_fun)
        |         set_digital_out(6,True)                     #Allumer la lumiere pour dire que l'on soude
        |         movej(tab_lin_deb_d[Index],a=a_fun,v=v_fun,t=t_fun,r=r_fun)
        | 
        |         fun_activer_soudure()                         #appel de la fonction activer la soudure
        | 
        |         movel(tab_lin_fin_d[Index],a=a_fun,v=vit_lin_d[Index],t=t_fun)
        | 
        |         fun_fin_soudure(2)                           #appel de la fonction désactiver la soudure
        | 
        |         movej(tab_lin_ret_d[Index],a=a_fun,v=v_fun,t=t_fun,r=r_fun)
        | 
        |         fun_deplacement_pose_inter(2)                     #appel de la fonction de déplacement en pose intermédiaire
        | 
        |     end
        |     sync()
        | end
      Script file /programs/Soudure 2023_03_27/V2.1/scripts/Execution/fun_soudure_point.script
        | def fun_soudure_point(Index,table):
        |     a_fun = 0.5
        |     v_fun = 1.1
        |     r_fun= 0.00
        |     t_fun = 0
        |     if (table == 1): #si 1 -> Table de gauche
        |         movej(tab_point_app_g[Index],a=a_fun,v=v_fun,t=t_fun,r= r_fun)
        |         set_digital_out(5,True)                     #Allumer la lumiere pour dire que l'on soude
        |         movej(tab_point_deb_g[Index],a=a_fun,v=v_fun,t=t_fun,r= r_fun)
        | 
        |         fun_activer_soudure()                         #appel de la fonction activer la soudure
        | 
        |         sleep(tps_point_g)                          #temps de soudure
        | 
        |         fun_fin_soudure(1)                           #appel de la fonction désactiver la soudure
        | 
        |         movej(tab_point_ret_g[Index],a=a_fun,v=v_fun,t=t_fun,r= r_fun)
        |         fun_deplacement_pose_inter(1)                     #appel de la fonction de déplacement en pose intermédiaire
        | 
        |     else: #sinon table de droite
        |         movej(tab_point_app_d[Index],a=a_fun,v=v_fun,t=t_fun,r= r_fun)
        |         set_digital_out(6,True)                     #Allumer la lumiere pour dire que l'on soude
        |         movej(tab_point_deb_d[Index],a=a_fun,v=v_fun,t=t_fun,r= r_fun)
        | 
        |         fun_activer_soudure()                         #appel de la fonction activer la soudure
        | 
        |         sleep(tps_point_d)                          #temps de soudure
        | 
        |         fun_fin_soudure(2)                           #appel de la fonction désactiver la soudure
        | 
        |         movej(tab_point_ret_d[Index],a=a_fun,v=v_fun,t=t_fun,r=r_fun)
        |         fun_deplacement_pose_inter(2)                     #appel de la fonction de déplacement en pose intermédiaire
        | 
        |     end
        |     sync()
        | end
    Folder Pas_A_Pas [hidden by the author, left out]
    Folder PopUps
      Folder Configuration [hidden by the author, left out]
      Folder Execution [hidden by the author, left out]
      Folder Pas_A_Pas [hidden by the author, left out]
Robot Program (runOnlyOnce=false)
  SuppressedNode
    Folder Initialisation
      Loop Counting (count=1) loopVariable(name=Boucle_10)
        Script: fun_adresse_bp()
  SuppressedNode
    MoveJ speed 60 deg/s, acceleration 80 deg/s^2 (useActiveTCP=true) feature=Base
      SafeHome (positionOptionType=SPEED_AND_ACCELERATION speed=1.047198 acceleration=1.396263 nextMotionTime=2)
      Waypoint PointPassage (Variable): motionParameters(jointSpeed=0.523599 jointAcceleration=0.698132 cartesianSpeed=0.25 cartesianAcceleration=1.2); variable(featureName=Point_init_G)
      Waypoint PointPassage (Variable): motionParameters(jointSpeed=0.523599 jointAcceleration=0.698132 cartesianSpeed=0.25 cartesianAcceleration=1.2); variable(featureName=Point_Attente_G)
      Waypoint PointPassage (Variable): motionParameters(jointSpeed=0.523599 jointAcceleration=0.698132 cartesianSpeed=0.25 cartesianAcceleration=1.2); variable(featureName=Point_config_g)
      Waypoint PointPassage (Variable): motionParameters(jointSpeed=0.523599 jointAcceleration=0.698132 cartesianSpeed=0.25 cartesianAcceleration=1.2); variable(featureName=Point_Attente_G)
      Waypoint PointPassage (Variable): motionParameters(jointSpeed=0.523599 jointAcceleration=0.698132 cartesianSpeed=0.25 cartesianAcceleration=1.2); variable(featureName=Point_init_G)
      SafeHome (positionOptionType=SPEED_AND_ACCELERATION speed=1.047198 acceleration=1.396263 nextMotionTime=2)
      Waypoint PointPassage (Variable): motionParameters(jointSpeed=0.785398 jointAcceleration=1.047198 cartesianSpeed=0.25 cartesianAcceleration=1.2); variable(featureName=Point_avt_initD)
      Waypoint PointPassage (Variable): motionParameters(jointSpeed=0.523599 jointAcceleration=0.698132 cartesianSpeed=0.25 cartesianAcceleration=1.2); variable(featureName=Point_init_D)
      Waypoint PointPassage (Variable): motionParameters(jointSpeed=0.523599 jointAcceleration=0.698132 cartesianSpeed=0.25 cartesianAcceleration=1.2); variable(featureName=Point_Attente_D)
      Waypoint PointPassage (Variable): motionParameters(jointSpeed=0.523599 jointAcceleration=0.698132 cartesianSpeed=0.25 cartesianAcceleration=1.2); variable(featureName=Point_config_d)
      Waypoint PointPassage (Variable): motionParameters(jointSpeed=0.523599 jointAcceleration=0.698132 cartesianSpeed=0.25 cartesianAcceleration=1.2); variable(featureName=Point_Attente_D)
      Waypoint PointPassage (Variable): motionParameters(jointSpeed=0.523599 jointAcceleration=0.698132 cartesianSpeed=0.25 cartesianAcceleration=1.2); variable(featureName=Point_init_D)
      SafeHome (positionOptionType=SPEED_AND_ACCELERATION speed=1.047198 acceleration=1.396263 nextMotionTime=2)
  safe_mode := 0
  Folder Deplacement vers position initial
    SuppressedNode
      Popup Message (haltProgram=false message=debut deplacement vers position initiale inputType=Text)
    Set DigitalOutput pin=Cmd_Carter_Bit1; digitalValue=0
    Set DigitalOutput pin=Cmd_Carter_Bit2; digitalValue=0
    Loop While (checkContinuously=false) expression=SecuGaucheOk≟ True  or SecuDroiteOk≟ True
      Script: sync()
      'clingottement pour signifier qu'il y  un defaut sur un des carters '
      Set DigitalOutput pin=Dcy_Voyant; digitalValue=0
      Set DigitalOutput pin=Led_Arret; digitalValue=0
      Wait Sleep waitTime=0.5
      Set DigitalOutput pin=Dcy_Voyant; digitalValue=1
      Set DigitalOutput pin=Led_Arret; digitalValue=1
      Wait Sleep waitTime=0.5
    Set DigitalOutput pin=Led_Arret; digitalValue=0
    Set DigitalOutput pin=Dcy_Voyant; digitalValue=0
    Wait Sleep waitTime=2
    'etre sur de l'ouverture complete du carter '
    MoveL speed 0.2 mm/s, acceleration 10 mm/s^2 (useActiveTCP=true) feature=Base
      Waypoint PointPassage_12 (Relative): relativeFromPosition TCP in base x=100.468 y=319.613 z=576.47 mm, rx=-0.0214 ry=-0.0122 rz=1.5415 rad; joints [-139.419, 75.739, -163.156, -3.26, 89.083, -42.172] deg; TCP offset x=-8.331 y=2.512 z=301.573 mm, rx=0 ry=0 rz=0 rad; TCP in base x=100.463 y=319.639 z=576.462 mm, rx=-0.0214 ry=-0.0122 rz=1.5416 rad; joints [-139.419, 75.741, -163.155, -3.263, 89.08, -42.17] deg
      'Pos_cobot a etait affectuer a la position init (l3)'
      'Pos_cobot[2] correspond a la valeur Z de la postion init (l4)'
    SuppressedNode
      MoveJ speed 60 deg/s, acceleration 80 deg/s^2 (useActiveTCP=true) feature=Base
        SuppressedNode
          Waypoint Position_init: motionParameters(jointSpeed=1.047198 jointAcceleration=1.396263 cartesianSpeed=0.25 cartesianAcceleration=1.2); TCP in base x=96.613 y=317.698 z=575.432 mm, rx=-0.0254 ry=-0.0254 rz=1.5393 rad; joints [-139.566, 75.575, -163.284, -3.665, 88.92, -42.143] deg; TCP offset x=-6.782 y=1.742 z=298.685 mm, rx=0 ry=0 rz=0 rad
        SuppressedNode
          Waypoint PointPassage (Variable): variable(featureName=Point_init)
        'Apres avoir eu la position du robot et tester la valeur de Z pour faire un mouvement verticale on envoi le robot en position init'
    angle_base := get_actual_joint_positions()
    If angle_base[0] ≤0.7
      If angle_base[0]≥1.6
        SafeHome (positionOptionType=SPEED_AND_ACCELERATION speed=1.047198 acceleration=1.396263 nextMotionTime=2)
      ElseIf angle_base[0]>1.6
        MoveJ speed 100 deg/s, acceleration 80 deg/s^2 (useActiveTCP=true) feature=Base
          Waypoint PointPassage (Variable): variable(featureName=Point_init_D)
          Waypoint PointPassage (Variable): variable(featureName=Point_avt_initD)
      ElseIf angle_base[0]<0.7
        MoveJ speed 100 deg/s, acceleration 80 deg/s^2 (useActiveTCP=true) feature=Base
          Waypoint PointPassage (Variable): variable(featureName=Point_init_G)
    ElseIf angle_base[0]>1.6
      MoveJ speed 100 deg/s, acceleration 80 deg/s^2 (useActiveTCP=true) feature=Base
        Waypoint PointPassage (Variable): variable(featureName=Point_init_D)
        Waypoint PointPassage (Variable): variable(featureName=Point_avt_initD)
    ElseIf angle_base[0]<0.7
      MoveJ speed 100 deg/s, acceleration 80 deg/s^2 (useActiveTCP=true) feature=Base
        Waypoint PointPassage (Variable): variable(featureName=Point_init_G)
    SafeHome (positionOptionType=SPEED_AND_ACCELERATION speed=1.047198 acceleration=1.396263 nextMotionTime=2)
    angle_base := get_actual_joint_positions()
  'mode config'
  If Mode_manu ≟ False  and config_reglage ≟ False
    If (config_g ≟ 1)  and  (config_d ≟ 1)
      Script: pop_up_config_g_et_d()
    ElseIf (config_g ≟1)
      Script: pop_up_config_g()
    ElseIf config_d ≟ 1
      Script: pop_up_config_d()
    ElseIf (config_g ≟ 0) and (config_d ≟ 0)
      Script: pop_up_config()
    boucle := 1
    Loop While (checkContinuously=false) expression=(Mode_manu ≟ False ) and (boucle ≟ 1)  and (config_reglage≟ False )
      Loop While (checkContinuously=true) expression=Pret_Table_Droi≟ False  and Pret_Table_Gauc≟ False  and Mode_manu ≟  False  and config_reglage≟ False
        Set DigitalOutput pin=Voyant_Table_Ga; digitalValue=1
        Set DigitalOutput pin=Voyant_Table_Dr; digitalValue=0
        Wait Sleep waitTime=0.5
        Set DigitalOutput pin=Voyant_Table_Ga; digitalValue=0
        Set DigitalOutput pin=Voyant_Table_Dr; digitalValue=1
        Wait Sleep waitTime=0.5
        Script: sync()
      If Pret_Table_Gauc ≟ True
        Set DigitalOutput pin=Voyant_Table_Ga; digitalValue=1
        Set DigitalOutput pin=Voyant_Table_Dr; digitalValue=0
        'plus de demande du nombre de point a saisir'
        MoveJ speed 60 deg/s, acceleration 80 deg/s^2 (useActiveTCP=true) feature=Base
          Waypoint PointPassage (Variable): motionParameters(blendRadius=0.006); variable(featureName=Point_init_G)
          Waypoint PointPassage (Variable): motionParameters(blendRadius=0.006); variable(featureName=Point_Attente_G)
          Waypoint PointPassage (Variable): motionParameters(jointSpeed=0.523599 jointAcceleration=0.698132 cartesianSpeed=0.25 cartesianAcceleration=1.2); variable(featureName=Point_config_g)
          led_cobot := 1
          Script: fun_config_g()
          led_cobot := 0
          Script: fun_valid_config_g()
          MoveJ speed 60 deg/s, acceleration 80 deg/s^2 (useActiveTCP=true) feature=Base
            SuppressedNode
              Waypoint anti_poq_g: motionParameters(jointSpeed=0.523599 jointAcceleration=0.698132 cartesianSpeed=0.25 cartesianAcceleration=1.2 blendRadius=0.07); TCP in base x=433.126 y=153.22 z=577.202 mm, rx=0.0572 ry=-0.0147 rz=1.5652 rad; joints [-179.123, 70.738, -150.145, -9.057, 92.825, -1.059] deg; TCP offset x=-8.331 y=2.512 z=301.573 mm, rx=0 ry=0 rz=0 rad
            Waypoint PointPassage (Variable): motionParameters(blendRadius=0.006); variable(featureName=Point_Attente_G)
            Waypoint PointPassage (Variable): motionParameters(blendRadius=0.006); variable(featureName=Point_init_G)
            SuppressedNode
              Waypoint PointPassage (Variable): motionParameters(jointSpeed=0.523599 jointAcceleration=0.698132 cartesianSpeed=0.25 cartesianAcceleration=1.2); variable(featureName=Point_init)
            SafeHome (positionOptionType=SPEED_AND_ACCELERATION speed=1.047198 acceleration=1.396263 nextMotionTime=2)
      If Pret_Table_Droi ≟ True
        Set DigitalOutput pin=Voyant_Table_Dr; digitalValue=1
        Set DigitalOutput pin=Voyant_Table_Ga; digitalValue=0
        MoveJ speed 60 deg/s, acceleration 80 deg/s^2 (useActiveTCP=true) feature=Base
          Waypoint PointPassage (Variable): motionParameters(blendRadius=0.006); variable(featureName=Point_avt_initD)
          Waypoint PointPassage (Variable): variable(featureName=Point_init_D)
          Waypoint PointPassage (Variable): motionParameters(blendRadius=0.006); variable(featureName=Point_Attente_D)
          Waypoint PointPassage (Variable): motionParameters(jointSpeed=0.523599 jointAcceleration=0.698132 cartesianSpeed=0.25 cartesianAcceleration=1.2); variable(featureName=Point_config_d)
        led_cobot := 1
        Script: fun_config_d()
        led_cobot := 0
        Script: fun_valid_config_d()
        MoveJ speed 60 deg/s, acceleration 80 deg/s^2 (useActiveTCP=true) feature=Base
          SuppressedNode
            Waypoint anti_poq_1_d: motionParameters(jointSpeed=0.523599 jointAcceleration=0.698132 cartesianSpeed=0.25 cartesianAcceleration=1.2 blendRadius=0); TCP in base x=-432.081 y=47.828 z=581.386 mm, rx=0.0024 ry=-0.0004 rz=1.5709 rad; joints [-31.202, 71.743, -153.151, -8.683, 90.121, -148.72] deg
          SuppressedNode
            Waypoint anti_poq_2_d: motionParameters(jointSpeed=1.047198 jointAcceleration=1.396263 cartesianSpeed=0.25 cartesianAcceleration=1.2 blendRadius=0.07); TCP in base x=-292.604 y=310.313 z=583.956 mm, rx=-0.0324 ry=-0.0877 rz=3.0963 rad; joints [-72.124, 71.739, -151.869, -12.519, 87.987, -20.279] deg; TCP offset x=-8.331 y=2.512 z=301.573 mm, rx=0 ry=0 rz=0 rad
          SuppressedNode
            Waypoint PointPassage (Variable): motionParameters(jointSpeed=0.785398 jointAcceleration=1.047198 cartesianSpeed=0.25 cartesianAcceleration=1.2); variable(featureName=Point_init)
          Waypoint PointPassage (Variable): motionParameters(blendRadius=0.006); variable(featureName=Point_Attente_D)
          Waypoint PointPassage (Variable): motionParameters(blendRadius=0.006); variable(featureName=Point_init_D)
          Waypoint PointPassage (Variable): motionParameters(blendRadius=0.006); variable(featureName=Point_avt_initD)
          SafeHome (positionOptionType=SPEED_AND_ACCELERATION speed=1.047198 acceleration=1.396263 nextMotionTime=2)
  '"Reg"'
  If Mode_manu ≟ False  and config_reglage ≟ True
    If (config_g ≟ 1)  and  (config_d ≟ 1)
      Script: pop_up_reg_gd()
      boucle := 1
    ElseIf config_g ≟ 1
      Script: pop_up_reg_gd()
      boucle := 1
    ElseIf config_d ≟ 1
      Script: pop_up_reg_d()
      boucle := 1
    Else 
      Script: close_popup()
      Loop While (checkContinuously=false) expression=config_reglage ≟ True
        Popup Error (haltProgram=false message=Aucune configuration n'est actuellement detectée. inputType=Text)
    boucle := 1
    Loop While (checkContinuously=false) expression=(Mode_manu ≟ False ) and (boucle ≟ 1)  and (config_reglage≟ True )
      Loop While (checkContinuously=true) expression=Pret_Table_Droi≟ False  and Pret_Table_Gauc≟ False  and Mode_manu ≟  False  and config_reglage ≟ True
        If config_g ≟ 1
          Set DigitalOutput pin=Voyant_Table_Ga; digitalValue=1
        If config_d ≟ 1
          Set DigitalOutput pin=Voyant_Table_Dr; digitalValue=1
        Wait Sleep waitTime=0.5
        Set DigitalOutput pin=Voyant_Table_Ga; digitalValue=0
        Set DigitalOutput pin=Voyant_Table_Dr; digitalValue=0
        Wait Sleep waitTime=0.5
      If Pret_Table_Gauc ≟ True
        safe_mode := 1
        Set DigitalOutput pin=Voyant_Table_Ga; digitalValue=1
        Set DigitalOutput pin=Voyant_Table_Dr; digitalValue=0
        MoveJ speed 60 deg/s, acceleration 80 deg/s^2 (useActiveTCP=true) feature=Base
          Waypoint PointPassage (Variable): motionParameters(blendRadius=0.006); variable(featureName=Point_init_G)
          Waypoint PointPassage (Variable): motionParameters(blendRadius=0.006); variable(featureName=Point_Attente_G)
          Waypoint PointPassage (Variable): motionParameters(jointSpeed=0.523599 jointAcceleration=0.698132 cartesianSpeed=0.25 cartesianAcceleration=1.2); variable(featureName=pose_inter_g)
        led_cobot := 1
        Script: fun_Pas_A_Pas_g()
        led_cobot := 0
        safe_mode := 0
        boucle := 0
      If Pret_Table_Droi ≟ True
        safe_mode := 1
        Set DigitalOutput pin=Voyant_Table_Dr; digitalValue=1
        Set DigitalOutput pin=Voyant_Table_Ga; digitalValue=0
        MoveJ speed 60 deg/s, acceleration 80 deg/s^2 (useActiveTCP=true) feature=Base
          Waypoint PointPassage (Variable): motionParameters(blendRadius=0.006); variable(featureName=Point_avt_initD)
          Waypoint PointPassage (Variable): motionParameters(blendRadius=0.006); variable(featureName=Point_init_D)
          Waypoint PointPassage (Variable): motionParameters(jointSpeed=0.523599 jointAcceleration=0.698132 cartesianSpeed=0.25 cartesianAcceleration=1.2); variable(featureName=pose_inter_d)
        led_cobot := 1
        Script: fun_Pas_A_Pas_d()
        led_cobot := 0
        safe_mode := 0
        boucle := 0
  'mode exe'
  If Mode_manu ≟ True
    If (config_g ≟ 1)  and  (config_d ≟ 1)
      Script: pop_up_exe()
      boucle := 1
    ElseIf config_g ≟ 1
      Script: pop_up_exe_g()
      boucle := 1
    ElseIf config_d ≟ 1
      Script: pop_up_exe_d()
      boucle := 1
    Else 
      Script: close_popup()
      Loop While (checkContinuously=false) expression=Mode_manu ≟ True
        Popup Error (haltProgram=false message=Aucune programmation n'est actuellement detectée, veillez à programmer une pièce avant de vouloir l'éxécuter. inputType=Text)
    Loop While (checkContinuously=false) expression=( Mode_manu ≟ True )  and (boucle ≟ 1)
      Loop While (checkContinuously=true) expression=Pret_Table_Droi≟ False  and Pret_Table_Gauc≟ False  and Mode_manu≟ True
        If config_g ≟ 1
          Set DigitalOutput pin=Voyant_Table_Ga; digitalValue=1
        If config_d ≟ 1
          Set DigitalOutput pin=Voyant_Table_Dr; digitalValue=1
        Wait Sleep waitTime=0.5
        Set DigitalOutput pin=Voyant_Table_Ga; digitalValue=0
        Set DigitalOutput pin=Voyant_Table_Dr; digitalValue=0
        Wait Sleep waitTime=0.5
      If (Pret_Table_Gauc ≟ True ) and (config_g ≟ True )
        boucle_g := 1
        SuppressedNode
          Script: pop_up_deb_exe_g()
        Loop While (checkContinuously=false) expression=boucle_g ≟ 1
          Set DigitalOutput pin=Cmd_Carter_Bit1; digitalValue=1
          Set DigitalOutput pin=Voyant_Table_Ga; digitalValue=1
          Set DigitalOutput pin=Voyant_Table_Dr; digitalValue=0
          Wait Sleep waitTime=0.25
          Set DigitalOutput pin=Voyant_Table_Ga; digitalValue=0
          Wait Sleep waitTime=0.25
          If SecuGaucheOk ≟  False
            Set DigitalOutput pin=Voyant_Table_Ga; digitalValue=1
            SuppressedNode
              Wait Sleep waitTime=6
            If SecuGaucheOk ≟  False
              Script: close_popup()
              Wait DigitalInput pin=SecuGaucheOk; digitalValue=1
          If SecuGaucheOk ≟  True
            secu_g := 1
            Set DigitalOutput pin=Voyant_Table_Ga; digitalValue=1
            MoveJ speed 60 deg/s, acceleration 80 deg/s^2 (useActiveTCP=true) feature=Base
              Waypoint PointPassage (Variable): motionParameters(blendRadius=0.006); variable(featureName=Point_init_G)
              SuppressedNode
                Waypoint PointPassage (Variable): motionParameters(blendRadius=0.006); variable(featureName=Point_Attente_G)
            Script: fun_execution_g()
            MoveJ speed 60 deg/s, acceleration 80 deg/s^2 (useActiveTCP=true) feature=Base
              Waypoint PointPassage (Variable): motionParameters(blendRadius=0.006); variable(featureName=Point_Attente_G)
              Waypoint PointPassage (Variable): motionParameters(blendRadius=0.006); variable(featureName=Point_init_G)
              SafeHome (positionOptionType=SPEED_AND_ACCELERATION speed=1.047198 acceleration=1.396263 nextMotionTime=2)
            Set DigitalOutput pin=Cmd_Carter_Bit1; digitalValue=0
            secu_g := 0
            boucle_g := 0
        boucle := 0
      ElseIf (Pret_Table_Gauc ≟ True ) and (config_g ≟ False )
        Script: close_popup()
        Popup Error (haltProgram=false message=Aucune programmation n'est actuellement detectée sur la table gauche, veillez à programmer une pièce avant de vouloir l'éxécuter. inputType=Text)
        boucle := 0
      If (Pret_Table_Droi ≟ True ) and (config_d ≟ True )
        boucle_d := 1
        Script: pop_up_deb_exe_d()
        Loop While (checkContinuously=false) expression=boucle_d ≟ 1
          Set DigitalOutput pin=Cmd_Carter_Bit2; digitalValue=1
          Set DigitalOutput pin=Voyant_Table_Ga; digitalValue=0
          Set DigitalOutput pin=Voyant_Table_Dr; digitalValue=1
          Wait Sleep waitTime=0.25
          Set DigitalOutput pin=Voyant_Table_Dr; digitalValue=0
          Wait Sleep waitTime=0.25
          If SecuDroiteOk ≟  False
            Set DigitalOutput pin=Voyant_Table_Dr; digitalValue=1
            Wait Sleep waitTime=6
            If SecuDroiteOk ≟  False
              Script: close_popup()
              Wait DigitalInput pin=SecuDroiteOk; digitalValue=1
          If SecuDroiteOk ≟  True
            secu_d := 1
            Set DigitalOutput pin=Voyant_Table_Dr; digitalValue=1
            MoveJ speed 60 deg/s, acceleration 80 deg/s^2 (useActiveTCP=true) feature=Base
              Waypoint PointPassage (Variable): variable(featureName=Point_avt_initD)
              SuppressedNode
                Waypoint PointPassage (Variable): motionParameters(blendRadius=0.006); variable(featureName=Point_init_D)
            Script: fun_execution_d()
            Set DigitalOutput pin=Cmd_Carter_Bit2; digitalValue=0
            secu_d := 0
            boucle_d := 0
        boucle := 0
      ElseIf (Pret_Table_Droi ≟ True ) and (config_d ≟ False )
        Script: close_popup()
        Popup Error (haltProgram=false message=Aucune programmation n'est actuellement detectée sur la table droite, veillez à programmer une pièce avant de vouloir l'éxécuter. inputType=Text)
        boucle := 0
Thread Thread_1 (runOnlyOnce=false)
  Folder Test_Ordre_Marche [hidden by the author, left out]
  Script: sync()
Thread Thread_2 (runOnlyOnce=false)
  Folder mode_soudure
    If Mode_soudure ≟  True
      If Mode_soudure≟ True  and soudure_on ≟ True
        fin_soud := 0
        Test_Ordre_Mar := True
        Test_Job := True
        Wait Condition expression=Test_Ordre_Mar≟ False
        Wait Condition expression=Test_Job≟ False
        Set DigitalOutput pin=Arc_On; digitalValue=1
        Test_Gaz := True
        'Test_Gaz permet de faire un appel dans le thread pour tester l'arriver gaz'
        Wait Condition expression=Valide_Gaz≟ True
        'Valide_Gaz permet  de connaitre quand le traitement de l'arriver gaz est terminer ans le thread.'
      ElseIf Mode_soudure ≟ True  and soudure_on ≟ False
        'Attente post debit gaz'
        Set DigitalOutput pin=Arc_On; digitalValue=0
        Test_Gaz := False
        Loop While (checkContinuously=false) expression=Reponse_Arc ≟ 1
          fin_soud := 0
          Script: sync()
        fin_soud := 1
  Script: sync()
Thread Thread_3 (runOnlyOnce=false)
  Folder led_cobot_2
    If led_cobot ≟ True
      If valider_bp_co ≟ True
        Set DigitalOutput pin=tool_out[1]; digitalValue=1
        Wait Sleep waitTime=0.25
        Set DigitalOutput pin=tool_out[1]; digitalValue=0
        Wait Sleep waitTime=0.25
        Set DigitalOutput pin=tool_out[1]; digitalValue=1
        Wait Sleep waitTime=0.25
        Set DigitalOutput pin=tool_out[1]; digitalValue=0
        Wait Sleep waitTime=0.25
        Set DigitalOutput pin=tool_out[1]; digitalValue=1
        Wait Sleep waitTime=0.25
        Set DigitalOutput pin=tool_out[1]; digitalValue=0
        Wait Sleep waitTime=0.25
        Script: sync()
      Script: sync()
    Script: sync()
  Script: sync()
Thread Thread_4 (runOnlyOnce=false)
  Folder led_cobot [hidden by the author, left out]
  Script: sync()
Thread Thread_5 (runOnlyOnce=false)
  Folder Test_Arc_On [hidden by the author, left out]
  Script: sync()
Thread Thread_6 (runOnlyOnce=false)
  Folder Test_Job
    If Test_Job≟ True
      SuppressedNode
        If Program_Soudure≟1 removedSiblings(If(type=ElseIf checkContinuously=false, expression=Program_Soudure≟2, children(Set(type=DigitalOutput, pin=Job_1, digitalValue=0), Set(type=DigitalOutput, pin=Job_2, digitalValue=1))), If(type=ElseIf checkContinuously=false, expression=Program_Soudure≟3, children(Set(type=DigitalOutput, pin=Job_1, digitalValue=1), Set(type=DigitalOutput, pin=Job_2, digitalValue=1))), If(type=ElseIf checkContinuously=false, expression=Program_Soudure≟4, children(Set(type=DigitalOutput, pin=Job_1, digitalValue=0), Set(type=DigitalOutput, pin=Job_2, digitalValue=0))), If(type=Else checkContinuously=false, children(Script(type=Line, expression=close_popup()), Popup(type=Error haltProgram=false message=Le Job soudure choisi n'existe pas. inputType=Text))))
          Set DigitalOutput pin=Job_1; digitalValue=1
          Set DigitalOutput pin=Job_2; digitalValue=0
      Test_Job := False
  Script: sync()
Thread Thread_7 (runOnlyOnce=false)
  Folder secu
    If SecuGaucheOk ≟  False  and secu_g ≟ 1
      Script: close_popup()
      Popup Error (haltProgram=true message=ATTENTION : Defaut carter ! inputType=Text)
    ElseIf SecuDroiteOk ≟ False  and secu_d ≟ 1
      Script: close_popup()
      Popup Error (haltProgram=true message=ATTENTION : Defaut carter ! inputType=Text)
  Script: sync()
Thread Thread_8 (runOnlyOnce=false)
  Folder bloq_soud_arret
    If Mode_soudure≟ False  and Test_Gaz ≟ True
      Script: close_popup()
      Popup Error (haltProgram=true message=Defaut : L'ordre de soudure a ete coupe pendant l'utilisation. inputType=Text)
  SuppressedNode
    Folder freedrive_droit
      If led_cobot ≟  True
        If tool_in[1] ≟ True
          Script: teach_mode()
        Else 
          Script: end_teach_mode()
  Script: sync()
SuppressedNode
  Thread Thread_9 (runOnlyOnce=false)
    Folder reglage
      If reglage_d ≠0
        Script file /programs/Programmes/cobot_v2/sript/Part_reglage/REGLAGE_D.script
          |     ##############################################################################
          | 
          | ########################soudure point#########################################
          | 
          |     ##############################################################################
          | 
          |         if reglage_d == 1:                                    #remplissage tableau
          |             teach_mode()
          |             fun_popup_soud(1, 1, i)
          |             fun_front_up(adresse_bp_cobot)
          |             tab_point_app_d[i] =  get_actual_tcp_pose()     #Enregistrer position dans tableau d'approche des soudue points quand appui bouton
          |             close_popup()
          | 
          |             fun_popup_soud(2, 1, i)
          |             fun_front_up(adresse_bp_cobot)
          |             tab_point_deb_d[i] =  get_actual_tcp_pose()     #Enregistrer position debut quand appui bouton bp_cobot
          |             close_popup()
          | 
          |             tab_point_ret_d[i] = tab_point_app_d[i]         #point de retrait est le meme que le point d approche
          |             end_teach_mode()
          |             global reconfig = 1
          |             global reglage_d = 0
          | 
          |             sync()
          | 
          |         ##############################################################################
          | 
          |     ##############################################################################
          | 
          | ########################soudure lineaire######################################
          | 
          |     ##############################################################################
          | 
          |         elif reglage_d == 2:                		            #remplissage tableau
          |             teach_mode()
          |             fun_popup_soud(1, 2, j)
          |             fun_front_up(adresse_bp_cobot)
          |             tab_lin_app_d[j] =  get_actual_tcp_pose()     	#Enregistrer position dans tableau d approche des soudures lineaire quand appui Bp_cobot
          |             close_popup()
          | 
          |             fun_popup_soud(2, 2, j)
          |             fun_front_up(adresse_bp_cobot)
          |             tab_lin_deb_d[j] =  get_actual_tcp_pose()     	#Enregistrer position dans tableau debut quand appui Bp_cobot
          |             close_popup()
          | 
          |             fun_popup_soud(6, 2, j)
          |             fun_front_up(adresse_bp_cobot)
          |             tab_lin_fin_d[j] =  get_actual_tcp_pose()     	#Enregistrer position dans un tableau fin quand appui Bp_cobot
          |             close_popup()
          | 
          |             vit_lin_d[j] = fun_demande_vit(2)
          | 
          |             fun_popup_soud(7, 2, j)
          |             fun_front_up(adresse_bp_cobot)
          |             tab_lin_ret_d[j] =  get_actual_tcp_pose()     	#Enregistrer position dans tableau retrait quand appui Bp_cobot
          |             close_popup()
          |             end_teach_mode()
          |             global reglage_d = 0
          | 
          |             sync()
          | 
          |         ##############################################################################
          | 
          |     ##############################################################################
          | 
          | #########################soudure arc de cercle##################################
          | 
          |     #################################################################################
          | 
          |         elif reglage_d == 3:                                  #remplissage tableau
          |             teach_mode()
          |             fun_popup_soud(1, 3, k)
          |             fun_front_up(adresse_bp_cobot)
          |             tab_arc_app_d[k] =  get_actual_tcp_pose() 	    #Enregistrer position dans tableau d approche des soudures arc de cercle quand appui
          |             close_popup()
          | 
          |             fun_popup_soud(2, 3, k)
          |             fun_front_up(adresse_bp_cobot)
          |             tab_arc_deb_d[k] =  get_actual_tcp_pose() 	    #Enregistrer position dans tableau debut quand appui Bp_d
          |             close_popup()
          | 
          |             fun_popup_soud(4, 3, k)
          |             fun_front_up(adresse_bp_cobot)
          |             tab_arc_mil_d[k] =  get_actual_tcp_pose() 	    #Enregistrer position dans tableau milieu quand appui Bp_cobot
          |             close_popup()
          | 
          |             fun_popup_soud(6, 3, k)
          |             fun_front_up(adresse_bp_cobot)
          |             tab_arc_fin_d[k] =  get_actual_tcp_pose() 	    #Enregistrer position dans un tableau fin quand appui Bp_cobot
          |             close_popup()
          | 
          |             vit_arc_d[k] = fun_demande_vit(3)               #demande de vitesse des soudures lineaire
          | 
          |             fun_popup_soud(7, 3, k)
          |             fun_front_up(adresse_bp_cobot)
          |             tab_arc_ret_d[k] =  get_actual_tcp_pose() 	    #Enregistrer position dans tableau retrait quand appui Bp_cobot
          |             close_popup()
          |             end_teach_mode()
          |             global reglage_d = 0
          | 
          |             sync()
          | 
          |         ##############################################################################
          | 
          |     ##############################################################################
          | 
          | ############################soudure cercle####################################
          | 
          |     #################################################################################
          | 
          |         elif reglage_d == 4:                                  #remplissage tableau
          |             teach_mode()
          |             fun_popup_soud(1, 4, l)
          |             fun_front_up(adresse_bp_cobot)
          |             tab_cer_app_d[l] =  get_actual_tcp_pose()     	#Enregistrer position dans tableau d approche des soudures arc de cercle quand appui Bp_cobot
          |             close_popup()
          | 
          |             fun_popup_soud(2, 4, l)
          |             fun_front_up(adresse_bp_cobot)
          |             tab_cer_deb_d[l] =  get_actual_tcp_pose()     	#Enregistrer position dans tableau debut quand appui Bp_cobot
          |             close_popup()
          | 
          |             fun_popup_soud(3, 4, l)
          |             fun_front_up(adresse_bp_cobot)
          |             tab_cer_quart_d[l] =  get_actual_tcp_pose()   	#Enregistrer position dans tableau d'approche des soudures arc de cercle quand appui Bp_d
          |             close_popup()
          | 
          |             fun_popup_soud(4, 4, l)
          |             fun_front_up(adresse_bp_cobot)
          |             tab_cer_mil_d[l] =  get_actual_tcp_pose()     	#Enregistrer position dans tableau milieu quand appui Bp_cobot
          |             close_popup()
          | 
          |             fun_popup_soud(5, 4, l)
          |             fun_front_up(adresse_bp_cobot)
          |             tab_cer_tro_d[l] =  get_actual_tcp_pose()     	#Enregistrer position dans tableau milieu quand appui Bp_cobot
          |             close_popup()
          | 
          |             fun_popup_soud(6, 4, l)
          |             fun_front_up(adresse_bp_cobot)
          |             tab_cer_fin_d[l] =  get_actual_tcp_pose()     	#Enregistrer position dans un tableau fin quand appui Bp_cobot
          |             close_popup()
          | 
          |             vit_cer_d[l] = fun_demande_vit(4)
          | 
          |             fun_popup_soud(7, 4, l)
          |             fun_front_up(adresse_bp_cobot)
          |             tab_cer_ret_d[l] =  get_actual_tcp_pose()    	#position de retrait est la meme que position d approche
          |             close_popup()
          |             end_teach_mode()
          |             global reglage_d = 0
          |             sync()
          | 
          |         end
          | 
          |     ##############################################################################
          | 
          | ############################################################
        Script: sync()
      If reglage_g ≠0
        Script file /programs/usbdisk_0/COBOT/finish/reg/REGLAGE_G.script
          |     ##############################################################################
          | 
          | ########################soudure point#########################################
          | 
          |     ##############################################################################
          | 
          |         if reglage_g == 1:                                    #remplissage tableau
          |             teach_mode()
          |             fun_popup_soud(1, 1, i)
          |             fun_front_up(adresse_bp_cobot)
          |             tab_point_app_g[i] =  get_actual_tcp_pose()     #Enregistrer position dans tableau d'approche des soudue points quand appui bouton
          |             close_popup()
          | 
          |             fun_popup_soud(2, 1, i)
          |             fun_front_up(adresse_bp_cobot)
          |             tab_point_deb_g[i] =  get_actual_tcp_pose()     #Enregistrer position debut quand appui bouton bp_cobot
          |             close_popup()
          | 
          |             tab_point_ret_g[i] = tab_point_app_g[i]         #point de retrait est le meme que le point d approche
          |             end_teach_mode()
          |             global reconfig = 1
          |             global reglage_g = 0
          | 
          |             sync()
          | 
          |         ##############################################################################
          | 
          |     ##############################################################################
          | 
          | ########################soudure lineaire######################################
          | 
          |     ##############################################################################
          | 
          |         elif reglage_g == 2:                		            #remplissage tableau
          |             teach_mode()
          |             fun_popup_soud(1, 2, j)
          |             fun_front_up(adresse_bp_cobot)
          |             tab_lin_app_g[j] =  get_actual_tcp_pose()     	#Enregistrer position dans tableau d approche des soudures lineaire quand appui Bp_cobot
          |             close_popup()
          | 
          |             fun_popup_soud(2, 2, j)
          |             fun_front_up(adresse_bp_cobot)
          |             tab_lin_deb_g[j] =  get_actual_tcp_pose()     	#Enregistrer position dans tableau debut quand appui Bp_cobot
          |             close_popup()
          | 
          |             fun_popup_soud(6, 2, j)
          |             fun_front_up(adresse_bp_cobot)
          |             tab_lin_fin_g[j] =  get_actual_tcp_pose()     	#Enregistrer position dans un tableau fin quand appui Bp_cobot
          |             close_popup()
          | 
          |             vit_lin_g[j] = fun_demande_vit(2)
          | 
          |             fun_popup_soud(7, 2, j)
          |             fun_front_up(adresse_bp_cobot)
          |             tab_lin_ret_g[j] =  get_actual_tcp_pose()     	#Enregistrer position dans tableau retrait quand appui Bp_cobot
          |             close_popup()
          |             end_teach_mode()
          |             global reglage_g = 0
          | 
          |             sync()
          | 
          |         ##############################################################################
          | 
          |     ##############################################################################
          | 
          | #########################soudure arc de cercle##################################
          | 
          |     #################################################################################
          | 
          |         elif reglage_g == 3:                                  #remplissage tableau
          |             teach_mode()
          |             fun_popup_soud(1, 3, k)
          |             fun_front_up(adresse_bp_cobot)
          |             tab_arc_app_g[k] =  get_actual_tcp_pose() 	    #Enregistrer position dans tableau d approche des soudures arc de cercle quand appui
          |             close_popup()
          | 
          |             fun_popup_soud(2, 3, k)
          |             fun_front_up(adresse_bp_cobot)
          |             tab_arc_deb_g[k] =  get_actual_tcp_pose() 	    #Enregistrer position dans tableau debut quand appui BP_cobot
          |             close_popup()
          | 
          |             fun_popup_soud(4, 3, k)
          |             fun_front_up(adresse_bp_cobot)
          |             tab_arc_mil_g[k] =  get_actual_tcp_pose() 	    #Enregistrer position dans tableau milieu quand appui Bp_cobot
          |             close_popup()
          | 
          |             fun_popup_soud(6, 3, k)
          |             fun_front_up(adresse_bp_cobot)
          |             tab_arc_fin_g[k] =  get_actual_tcp_pose() 	    #Enregistrer position dans un tableau fin quand appui Bp_cobot
          |             close_popup()
          | 
          |             vit_arc_g[k] = fun_demande_vit(3)               #demande de vitesse des soudures lineaire
          | 
          |             fun_popup_soud(7, 3, k)
          |             fun_front_up(adresse_bp_cobot)
          |             tab_arc_ret_g[k] =  get_actual_tcp_pose() 	    #Enregistrer position dans tableau retrait quand appui Bp_cobot
          |             close_popup()
          |             end_teach_mode()
          |             global reglage_g = 0
          | 
          |             sync()
          | 
          |         ##############################################################################
          | 
          |     ##############################################################################
          | 
          | ############################soudure cercle####################################
          | 
          |     #################################################################################
          | 
          |         elif reglage_g == 4:                                  #remplissage tableau
          |             teach_mode()
          |             fun_popup_soud(1, 4, l)
          |             fun_front_up(adresse_bp_cobot)
          |             tab_cer_app_g[l] =  get_actual_tcp_pose()     	#Enregistrer position dans tableau d approche des soudures arc de cercle quand appui Bp_cobot
          |             close_popup()
          | 
          |             fun_popup_soud(2, 4, l)
          |             fun_front_up(adresse_bp_cobot)
          |             tab_cer_deb_g[l] =  get_actual_tcp_pose()     	#Enregistrer position dans tableau debut quand appui Bp_cobot
          |             close_popup()
          | 
          |             fun_popup_soud(3, 4, l)
          |             fun_front_up(adresse_bp_cobot)
          |             tab_cer_quart_g[l] =  get_actual_tcp_pose()   	#Enregistrer position dans tableau d'approche des soudures arc de cercle quand appui Bp_cobot
          |             close_popup()
          | 
          |             fun_popup_soud(4, 4, l)
          |             fun_front_up(adresse_bp_cobot)
          |             tab_cer_mil_g[l] =  get_actual_tcp_pose()     	#Enregistrer position dans tableau milieu quand appui Bp_cobot
          |             close_popup()
          | 
          |             fun_popup_soud(5, 4, l)
          |             fun_front_up(adresse_bp_cobot)
          |             tab_cer_tro_g[l] =  get_actual_tcp_pose()     	#Enregistrer position dans tableau milieu quand appui Bp_cobot
          |             close_popup()
          | 
          |             fun_popup_soud(6, 4, l)
          |             fun_front_up(adresse_bp_cobot)
          |             tab_cer_fin_g[l] =  get_actual_tcp_pose()     	#Enregistrer position dans un tableau fin quand appui Bp_cobot
          |             close_popup()
          | 
          |             vit_cer_g[l] = fun_demande_vit(4)
          | 
          |             fun_popup_soud(7, 4, l)
          |             fun_front_up(adresse_bp_cobot)
          |             tab_cer_ret_g[l] =  get_actual_tcp_pose()    	#position de retrait est la meme que position d approche
          |             close_popup()
          |             end_teach_mode()
          |             global reglage_g = 0
          |             sync()
          | 
          |         end
          | 
          |     ##############################################################################
          | 
          | ############################################################
        Script: sync()
      Script: sync()
    Script: sync()
Thread Thread_10 (runOnlyOnce=false)
  Folder reglage
    If safe_mode ≟ 1  and Mode_manu ≟  True
      Script: close_popup()
      Popup Error (haltProgram=true message=STOP !!!! inputType=Text)
    Script: sync()
  Script: sync()
